// Mitsubishi GX Works2 project: 240423_순위별우선회로   PLC: Q03UDV

PROGRAM MAIN
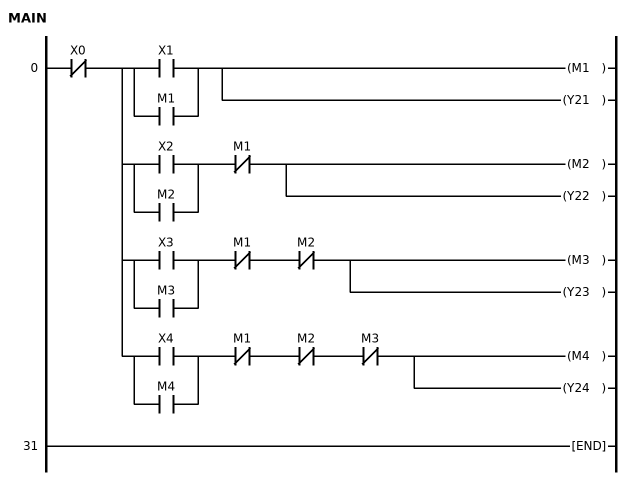
0     LDI     X0
      MPS
      LD      X1
      OR      M1
      ANB
      OUT     M1
      OUT     Y21
      MRD
      LD      X2
      OR      M2
      ANB
      ANI     M1
      OUT     M2
      OUT     Y22
      MRD
      LD      X3
      OR      M3
      ANB
      ANI     M1
      ANI     M2
      OUT     M3
      OUT     Y23
      MPP
      LD      X4
      OR      M4
      ANB
      ANI     M1
      ANI     M2
      ANI     M3
      OUT     M4
      OUT     Y24
31    END
END_PROGRAM
